// Mitsubishi GX Works2 project: Fan off delay   PLC: FX1N/FX1NC

PROGRAM MAIN
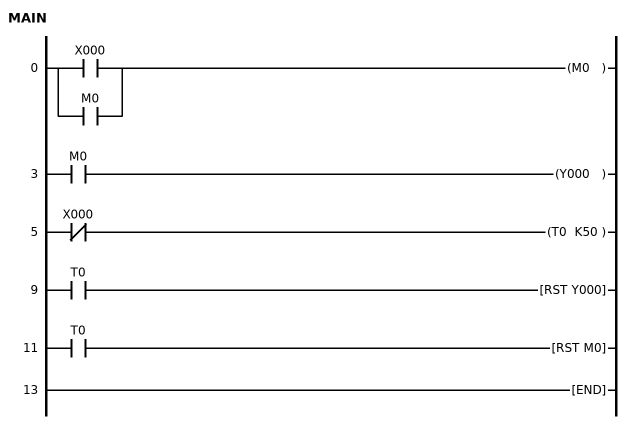
0     LD      X000
      OR      M0
      OUT     M0
3     LD      M0
      OUT     Y000
5     LDI     X000
      OUT     T0 K50
9     LD      T0
      RST     Y000
11    LD      T0
      RST     M0
13    END
END_PROGRAM
